// TIA Portal V17 export
// export: Created 2026-07-30T06:00:00.0000000Z, ExportSetting WithDefaults
FUNCTION "SclAssign" : Void   // FC10, SCL
VERSION : 0.1
// stored: AutoNumber true, IsIECCheckEnabled false
BEGIN

REGION Network 1: Write counters
   "GlobalData".Count := "GlobalData".Ready;
   "GlobalData".Config.MaxSpeed := "GlobalData".Count;
END_REGION

REGION Network 2: Gate ready flag
   IF "GlobalData".Config.Enabled THEN
   "GlobalData".Ready := FALSE;
   END_IF;
END_REGION
END_FUNCTION
